FUNCTION_BLOCK FB_PT100_EL3214 IMPLEMENTS I_TemperatureSensor
VAR_INPUT
END_VAR
VAR_OUTPUT
END_VAR
VAR
	//Property Real value
	fTemperature : REAL;
	//Raw value
	TempRaw AT %I* : INT;
	//Convertion parameters
	m : REAL := 0.1; //Multiplier for convertion
END_VAR

//Temperature measurement: PT 100 1/10 DIN + EL3214: 3-wire

PROPERTY Temperature : REAL
GET
fTemperature := INT_TO_REAL(TempRaw) * m;
Temperature := THIS^.fTemperature;
END_GET
END_PROPERTY

END_FUNCTION_BLOCK

(* stored: Version 1.1.0.1
   POU FB_PT100_EL3214: Id {53f33390-605b-45f3-b0c4-f896ba7505ff}, SpecialFunc None
   Property Temperature: Id {667d44b9-225d-41ed-bc93-6540bd10ff8f}
   Get Get: Id {041db4e0-f07a-4a4d-a863-73886e1b9200} *)
